Fanuc KAREL source: CLR_IO_STAT.kl

PROGRAM T
%NOLOCKGROUP
VAR
 v0 : FILE
BEGIN
 CLR_IO_STAT(v0)
END T
